ABB RAPID module: MainModule.mod

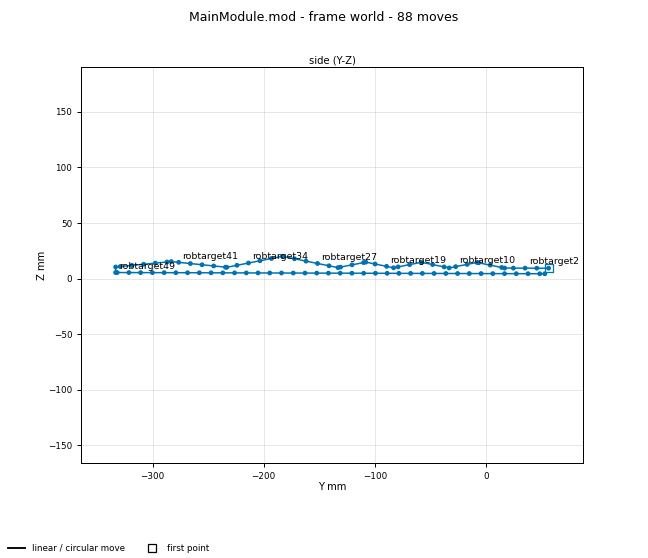
[picture p0: tool path of MainModule.mod in frame world, 88 of 89 moves have a stored position in this frame; points joined in program order, loops and branches not executed]
Module MainModule
!Declarations
!jointtarget
VAR jointtarget In:=[[7.408424,53.50812,4.795727,0.087915,31.638713,125.775488],[9E9,9E9,9E9,9E9,9E9,9E9]];

!robtarget
CONST robtarget robtarget0:=[[431.569187,56.285063,9.381984],[-0.000698,0.99784,0.064795,0.010754],[0,0,1,0],[9E9,9E9,9E9,9E9,9E9,9E9]];
CONST robtarget robtarget1:=[[431.569187,45.724144,9.412298],[-0.000572,0.998549,0.05275,0.010827],[0,0,1,0],[9E9,9E9,9E9,9E9,9E9,9E9]];
CONST robtarget robtarget2:=[[431.569187,35.163224,9.442612],[-0.000443,0.999115,0.040635,0.010893],[0,0,1,0],[9E9,9E9,9E9,9E9,9E9,9E9]];
CONST robtarget robtarget3:=[[431.569187,24.602305,9.472927],[-0.000312,0.999535,0.028467,0.010951],[0,0,1,0],[9E9,9E9,9E9,9E9,9E9,9E9]];
CONST robtarget robtarget4:=[[431.569187,16.862962,9.495142],[-0.000215,0.999749,0.019524,0.010988],[0,0,1,0],[9E9,9E9,9E9,9E9,9E9,9E9]];
CONST robtarget robtarget5:=[[431.569187,14.097751,10.056362],[-0.00019,0.999799,0.016325,0.011641],[0,-1,1,0],[9E9,9E9,9E9,9E9,9E9,9E9]];
CONST robtarget robtarget6:=[[431.569187,3.747803,12.15696],[-0.000061,0.999891,0.004342,0.01408],[0,-1,1,0],[9E9,9E9,9E9,9E9,9E9,9E9]];
CONST robtarget robtarget7:=[[431.569187,-6.602145,14.257559],[0.000126,0.999834,-0.007647,0.016509],[-1,0,1,0],[9E9,9E9,9E9,9E9,9E9,9E9]];
CONST robtarget robtarget8:=[[431.569187,-8.128353,14.567314],[0.000159,0.999813,-0.009415,0.016866],[-1,0,1,0],[9E9,9E9,9E9,9E9,9E9,9E9]];
CONST robtarget robtarget9:=[[431.569187,-16.962196,12.826988],[0.000292,0.999697,-0.019638,0.014842],[-1,0,1,0],[9E9,9E9,9E9,9E9,9E9,9E9]];
CONST robtarget robtarget10:=[[431.569187,-27.323994,10.785644],[0.000394,0.999423,-0.031607,0.012462],[-1,0,1,0],[9E9,9E9,9E9,9E9,9E9,9E9]];
CONST robtarget robtarget11:=[[431.569187,-33.145913,9.638687],[0.000427,0.999204,-0.038315,0.011124],[-1,0,1,0],[9E9,9E9,9E9,9E9,9E9,9E9]];
CONST robtarget robtarget12:=[[431.569187,-37.6806,10.559035],[0.00053,0.998978,-0.043528,0.012173],[-1,-1,1,0],[9E9,9E9,9E9,9E9,9E9,9E9]];
CONST robtarget robtarget13:=[[431.569187,-48.030548,12.659634],[0.000807,0.998359,-0.055384,0.01455],[-1,-1,1,0],[9E9,9E9,9E9,9E9,9E9,9E9]];
CONST robtarget robtarget14:=[[431.569187,-58.137228,14.71086],[0.00113,0.997617,-0.066893,0.016846],[-1,0,1,0],[9E9,9E9,9E9,9E9,9E9,9E9]];
CONST robtarget robtarget15:=[[431.569187,-58.380774,14.66288],[0.00113,0.9976,-0.06717,0.016789],[-1,0,1,0],[9E9,9E9,9E9,9E9,9E9,9E9]];
CONST robtarget robtarget16:=[[431.569187,-68.742572,12.621536],[0.001139,0.996779,-0.078889,0.014391],[-1,0,1,0],[9E9,9E9,9E9,9E9,9E9,9E9]];
CONST robtarget robtarget17:=[[431.569187,-79.10437,10.580192],[0.001091,0.995823,-0.090511,0.012005],[-1,0,1,0],[9E9,9E9,9E9,9E9,9E9,9E9]];
CONST robtarget robtarget18:=[[431.569187,-83.154788,9.782233],[0.001057,0.995413,-0.095024,0.011076],[-1,0,1,0],[9E9,9E9,9E9,9E9,9E9,9E9]];
CONST robtarget robtarget19:=[[431.569187,-89.45895,11.061709],[0.00128,0.994704,-0.102011,0.01248],[-1,-1,1,0],[9E9,9E9,9E9,9E9,9E9,9E9]];
CONST robtarget robtarget20:=[[431.569187,-99.808898,13.162308],[0.001684,0.993441,-0.11338,0.014757],[-1,-1,1,0],[9E9,9E9,9E9,9E9,9E9,9E9]];
CONST robtarget robtarget21:=[[431.569187,-108.146103,14.854406],[0.002043,0.992336,-0.122441,0.016561],[-1,0,1,0],[9E9,9E9,9E9,9E9,9E9,9E9]];
CONST robtarget robtarget22:=[[431.569187,-110.16115,14.457428],[0.002022,0.992072,-0.124619,0.016097],[-1,0,1,0],[9E9,9E9,9E9,9E9,9E9,9E9]];
CONST robtarget robtarget23:=[[431.569187,-120.522948,12.416084],[0.00188,0.990649,-0.135731,0.013723],[-1,0,1,0],[9E9,9E9,9E9,9E9,9E9,9E9]];
CONST robtarget robtarget24:=[[431.569187,-130.884746,10.37474],[0.001687,0.989116,-0.146689,0.011376],[-1,0,1,0],[9E9,9E9,9E9,9E9,9E9,9E9]];
CONST robtarget robtarget25:=[[431.569187,-133.163663,9.925778],[0.001638,0.988764,-0.149077,0.010864],[-1,0,1,0],[9E9,9E9,9E9,9E9,9E9,9E9]];
CONST robtarget robtarget26:=[[431.569187,-141.2373,11.564383],[0.002005,0.987442,-0.157468,0.012572],[-1,-1,1,0],[9E9,9E9,9E9,9E9,9E9,9E9]];
CONST robtarget robtarget27:=[[431.569187,-151.587248,13.664982],[0.00251,0.985662,-0.168072,0.01472],[-1,-1,1,0],[9E9,9E9,9E9,9E9,9E9,9E9]];
CONST robtarget robtarget28:=[[431.569187,-161.937196,15.76558],[0.003052,0.983792,-0.178497,0.016819],[-1,-1,1,0],[9E9,9E9,9E9,9E9,9E9,9E9]];
CONST robtarget robtarget29:=[[431.569187,-172.287145,17.866179],[0.003627,0.981839,-0.188739,0.018868],[-1,-1,1,0],[9E9,9E9,9E9,9E9,9E9,9E9]];
CONST robtarget robtarget30:=[[431.569187,-182.637093,19.966778],[0.004233,0.979811,-0.19879,0.020864],[-1,0,1,0],[9E9,9E9,9E9,9E9,9E9,9E9]];
CONST robtarget robtarget31:=[[431.569187,-183.146294,20.070124],[0.004264,0.979709,-0.19928,0.020961],[-1,0,1,0],[9E9,9E9,9E9,9E9,9E9,9E9]];
CONST robtarget robtarget32:=[[431.569187,-192.998307,18.129211],[0.004,0.977797,-0.208678,0.018741],[-1,0,1,0],[9E9,9E9,9E9,9E9,9E9,9E9]];
CONST robtarget robtarget33:=[[431.569187,-203.360105,16.087868],[0.003681,0.97572,-0.21837,0.016447],[-1,0,1,0],[9E9,9E9,9E9,9E9,9E9,9E9]];
CONST robtarget robtarget34:=[[431.569187,-213.721903,14.046524],[0.003322,0.973584,-0.227864,0.014195],[-1,0,1,0],[9E9,9E9,9E9,9E9,9E9,9E9]];
CONST robtarget robtarget35:=[[431.569187,-224.083701,12.00518],[0.002927,0.971393,-0.237157,0.011989],[-1,0,1,0],[9E9,9E9,9E9,9E9,9E9,9E9]];
CONST robtarget robtarget36:=[[431.569187,-233.181413,10.21287],[0.002552,0.96943,-0.245149,0.010091],[-1,0,1,0],[9E9,9E9,9E9,9E9,9E9,9E9]];
CONST robtarget robtarget37:=[[431.569187,-234.46303,10.344732],[0.002593,0.969146,-0.246261,0.010205],[-1,0,1,0],[9E9,9E9,9E9,9E9,9E9,9E9]];
CONST robtarget robtarget38:=[[431.569187,-244.968535,11.425619],[0.002938,0.966803,-0.255262,0.011128],[-1,-1,1,0],[9E9,9E9,9E9,9E9,9E9,9E9]];
CONST robtarget robtarget39:=[[431.569187,-255.474039,12.506506],[0.003292,0.964427,-0.264055,0.012023],[-1,0,1,0],[9E9,9E9,9E9,9E9,9E9,9E9]];
CONST robtarget robtarget40:=[[431.569187,-265.979544,13.587392],[0.003653,0.962023,-0.272641,0.01289],[-1,0,1,0],[9E9,9E9,9E9,9E9,9E9,9E9]];
CONST robtarget robtarget41:=[[431.569187,-276.485048,14.668279],[0.00402,0.959595,-0.281021,0.013728],[-1,0,1,0],[9E9,9E9,9E9,9E9,9E9,9E9]];
CONST robtarget robtarget42:=[[431.569187,-283.177166,15.356815],[0.004257,0.958039,-0.286252,0.014248],[-1,0,1,0],[9E9,9E9,9E9,9E9,9E9,9E9]];
CONST robtarget robtarget43:=[[431.569187,-286.99274,14.986344],[0.00418,0.957159,-0.289201,0.013835],[-1,0,1,0],[9E9,9E9,9E9,9E9,9E9,9E9]];
CONST robtarget robtarget44:=[[431.569187,-297.504272,13.965734],[0.003958,0.954726,-0.297187,0.012716],[-1,0,1,0],[9E9,9E9,9E9,9E9,9E9,9E9]];
CONST robtarget robtarget45:=[[431.569187,-308.015803,12.945123],[0.003722,0.952283,-0.304974,0.011623],[-1,0,1,0],[9E9,9E9,9E9,9E9,9E9,9E9]];
CONST robtarget robtarget46:=[[431.569187,-318.527335,11.924513],[0.003474,0.949832,-0.312563,0.010557],[-1,0,1,0],[9E9,9E9,9E9,9E9,9E9,9E9]];
CONST robtarget robtarget47:=[[431.569187,-329.038866,10.903902],[0.003214,0.947378,-0.319958,0.009516],[-1,0,1,0],[9E9,9E9,9E9,9E9,9E9,9E9]];
CONST robtarget robtarget48:=[[431.569187,-333.199163,10.499961],[0.003108,0.946407,-0.322833,0.009112],[-1,0,1,0],[9E9,9E9,9E9,9E9,9E9,9E9]];
CONST robtarget robtarget49:=[[431.569187,-333.212285,5.499561],[0.001628,0.946436,-0.322853,0.004773],[-1,0,1,0],[9E9,9E9,9E9,9E9,9E9,9E9]];
CONST robtarget robtarget50:=[[431.569187,-331.831606,5.495597],[0.001625,0.946759,-0.321902,0.004779],[-1,0,1,0],[9E9,9E9,9E9,9E9,9E9,9E9]];
CONST robtarget robtarget51:=[[431.569187,-321.270687,5.465283],[0.001597,0.949235,-0.314526,0.004821],[-1,0,1,0],[9E9,9E9,9E9,9E9,9E9,9E9]];
CONST robtarget robtarget52:=[[431.569187,-310.709767,5.434969],[0.001569,0.95171,-0.306955,0.004863],[-1,0,1,0],[9E9,9E9,9E9,9E9,9E9,9E9]];
CONST robtarget robtarget53:=[[431.569187,-300.148848,5.404655],[0.001538,0.954181,-0.299186,0.004905],[-1,0,1,0],[9E9,9E9,9E9,9E9,9E9,9E9]];
CONST robtarget robtarget54:=[[431.569187,-289.587928,5.374341],[0.001506,0.956643,-0.291217,0.004946],[-1,0,1,0],[9E9,9E9,9E9,9E9,9E9,9E9]];
CONST robtarget robtarget55:=[[431.569187,-279.027009,5.344027],[0.001472,0.959093,-0.283043,0.004987],[-1,0,1,0],[9E9,9E9,9E9,9E9,9E9,9E9]];
CONST robtarget robtarget56:=[[431.569187,-268.466089,5.313713],[0.001436,0.961526,-0.274664,0.005026],[-1,0,1,0],[9E9,9E9,9E9,9E9,9E9,9E9]];
CONST robtarget robtarget57:=[[431.569187,-257.90517,5.283399],[0.001398,0.963937,-0.266078,0.005065],[-1,0,1,0],[9E9,9E9,9E9,9E9,9E9,9E9]];
CONST robtarget robtarget58:=[[431.569187,-247.34425,5.253085],[0.001358,0.966322,-0.257283,0.005102],[-1,0,1,0],[9E9,9E9,9E9,9E9,9E9,9E9]];
CONST robtarget robtarget59:=[[431.569187,-236.783331,5.222771],[0.001317,0.968674,-0.248278,0.005139],[-1,0,1,0],[9E9,9E9,9E9,9E9,9E9,9E9]];
CONST robtarget robtarget60:=[[431.569187,-226.222411,5.192457],[0.001274,0.970989,-0.239063,0.005173],[-1,0,1,0],[9E9,9E9,9E9,9E9,9E9,9E9]];
CONST robtarget robtarget61:=[[431.569187,-215.661492,5.162143],[0.001229,0.973261,-0.229639,0.005207],[-1,0,1,0],[9E9,9E9,9E9,9E9,9E9,9E9]];
CONST robtarget robtarget62:=[[431.569187,-205.100572,5.131828],[0.001181,0.975484,-0.220006,0.005238],[-1,0,1,0],[9E9,9E9,9E9,9E9,9E9,9E9]];
CONST robtarget robtarget63:=[[431.569187,-194.539653,5.101514],[0.001132,0.977651,-0.210166,0.005268],[-1,0,1,0],[9E9,9E9,9E9,9E9,9E9,9E9]];
CONST robtarget robtarget64:=[[431.569187,-183.978733,5.0712],[0.001082,0.979756,-0.200123,0.005295],[-1,0,1,0],[9E9,9E9,9E9,9E9,9E9,9E9]];
CONST robtarget robtarget65:=[[431.569187,-173.417814,5.040886],[0.001029,0.981793,-0.189879,0.00532],[-1,0,1,0],[9E9,9E9,9E9,9E9,9E9,9E9]];
CONST robtarget robtarget66:=[[431.569187,-162.856894,5.010572],[0.000975,0.983754,-0.179439,0.005343],[-1,0,1,0],[9E9,9E9,9E9,9E9,9E9,9E9]];
CONST robtarget robtarget67:=[[431.569187,-152.295975,4.980258],[0.000918,0.985634,-0.168808,0.005363],[-1,0,1,0],[9E9,9E9,9E9,9E9,9E9,9E9]];
CONST robtarget robtarget68:=[[431.569187,-141.735055,4.949944],[0.000861,0.987425,-0.157993,0.00538],[-1,0,1,0],[9E9,9E9,9E9,9E9,9E9,9E9]];
CONST robtarget robtarget69:=[[431.569187,-131.174136,4.91963],[0.000802,0.989121,-0.147,0.005394],[-1,0,1,0],[9E9,9E9,9E9,9E9,9E9,9E9]];
CONST robtarget robtarget70:=[[431.569187,-120.613216,4.889316],[0.000741,0.990716,-0.135838,0.005405],[-1,0,1,0],[9E9,9E9,9E9,9E9,9E9,9E9]];
CONST robtarget robtarget71:=[[431.569187,-110.052297,4.859002],[0.000679,0.992203,-0.124516,0.005412],[-1,0,1,0],[9E9,9E9,9E9,9E9,9E9,9E9]];
CONST robtarget robtarget72:=[[431.569187,-99.491377,4.828688],[0.000616,0.993575,-0.113044,0.005416],[-1,0,1,0],[9E9,9E9,9E9,9E9,9E9,9E9]];
CONST robtarget robtarget73:=[[431.569187,-88.930458,4.798373],[0.000552,0.994827,-0.101433,0.005416],[-1,0,1,0],[9E9,9E9,9E9,9E9,9E9,9E9]];
CONST robtarget robtarget74:=[[431.569187,-78.369538,4.768059],[0.000487,0.995954,-0.089695,0.005413],[-1,0,1,0],[9E9,9E9,9E9,9E9,9E9,9E9]];
CONST robtarget robtarget75:=[[431.569187,-67.808619,4.737745],[0.000422,0.996951,-0.077843,0.005406],[-1,0,1,0],[9E9,9E9,9E9,9E9,9E9,9E9]];
CONST robtarget robtarget76:=[[431.569187,-57.247699,4.707431],[0.000356,0.997812,-0.065891,0.005395],[-1,0,1,0],[9E9,9E9,9E9,9E9,9E9,9E9]];
CONST robtarget robtarget77:=[[431.569187,-46.68678,4.677117],[0.00029,0.998534,-0.053853,0.005379],[-1,0,1,0],[9E9,9E9,9E9,9E9,9E9,9E9]];
CONST robtarget robtarget78:=[[431.569187,-36.12586,4.646803],[0.000224,0.999114,-0.041744,0.00536],[-1,0,1,0],[9E9,9E9,9E9,9E9,9E9,9E9]];
CONST robtarget robtarget79:=[[431.569187,-25.564941,4.616489],[0.000158,0.999548,-0.029579,0.005337],[-1,0,1,0],[9E9,9E9,9E9,9E9,9E9,9E9]];
CONST robtarget robtarget80:=[[431.569187,-15.004022,4.586175],[0.000092,0.999835,-0.017375,0.005309],[-1,0,1,0],[9E9,9E9,9E9,9E9,9E9,9E9]];
CONST robtarget robtarget81:=[[431.569187,-4.443102,4.555861],[0.000027,0.999973,-0.005147,0.005278],[-1,0,1,0],[9E9,9E9,9E9,9E9,9E9,9E9]];
CONST robtarget robtarget82:=[[431.569187,6.117817,4.525547],[-0.000037,0.999961,0.007087,0.005242],[0,0,1,0],[9E9,9E9,9E9,9E9,9E9,9E9]];
CONST robtarget robtarget83:=[[431.569187,16.678737,4.495233],[-0.000101,0.9998,0.019312,0.005203],[0,0,1,0],[9E9,9E9,9E9,9E9,9E9,9E9]];
CONST robtarget robtarget84:=[[431.569187,27.239656,4.464919],[-0.000163,0.99949,0.031511,0.00516],[0,0,1,0],[9E9,9E9,9E9,9E9,9E9,9E9]];
CONST robtarget robtarget85:=[[431.569187,37.800576,4.434604],[-0.000223,0.999033,0.043668,0.005113],[0,0,1,0],[9E9,9E9,9E9,9E9,9E9,9E9]];
CONST robtarget robtarget86:=[[431.569187,48.361495,4.40429],[-0.000283,0.998431,0.055767,0.005063],[0,0,1,0],[9E9,9E9,9E9,9E9,9E9,9E9]];
CONST robtarget robtarget87:=[[431.569187,52.881866,4.391315],[-0.000308,0.99813,0.060925,0.00504],[0,0,1,0],[9E9,9E9,9E9,9E9,9E9,9E9]];

!speeddata
VAR speeddata speeddata0:=[250,572.957795,5000,1000];

!tooldata
PERS tooldata ToolOfLove:=[True,[[0.015258,-0.149222,99.918848],[1,0,0,0]],[0.001,[0,0,0.1],[1,0,0,0],0,0,0]];

!wobjdata
PERS wobjdata Root:=[False,True,"",[[0,0,0],[1,0,0,0]],[[0,0,0],[1,0,0,0]]];

!zonedata
VAR zonedata zonedata0:=[False,1,5,1,5,1,5];

Proc Main()
ConfL \On;
ConfJ \On;
SingArea \Wrist;
MoveAbsJ In, speeddata0, zonedata0, ToolOfLove;
MoveL robtarget0, speeddata0, zonedata0, ToolOfLove \WObj:=Root;
MoveL robtarget1, speeddata0, zonedata0, ToolOfLove \WObj:=Root;
MoveL robtarget2, speeddata0, zonedata0, ToolOfLove \WObj:=Root;
MoveL robtarget3, speeddata0, zonedata0, ToolOfLove \WObj:=Root;
MoveL robtarget4, speeddata0, zonedata0, ToolOfLove \WObj:=Root;
MoveL robtarget5, speeddata0, zonedata0, ToolOfLove \WObj:=Root;
MoveL robtarget6, speeddata0, zonedata0, ToolOfLove \WObj:=Root;
MoveL robtarget7, speeddata0, zonedata0, ToolOfLove \WObj:=Root;
MoveL robtarget8, speeddata0, zonedata0, ToolOfLove \WObj:=Root;
MoveL robtarget9, speeddata0, zonedata0, ToolOfLove \WObj:=Root;
MoveL robtarget10, speeddata0, zonedata0, ToolOfLove \WObj:=Root;
MoveL robtarget11, speeddata0, zonedata0, ToolOfLove \WObj:=Root;
MoveL robtarget12, speeddata0, zonedata0, ToolOfLove \WObj:=Root;
MoveL robtarget13, speeddata0, zonedata0, ToolOfLove \WObj:=Root;
MoveL robtarget14, speeddata0, zonedata0, ToolOfLove \WObj:=Root;
MoveL robtarget15, speeddata0, zonedata0, ToolOfLove \WObj:=Root;
MoveL robtarget16, speeddata0, zonedata0, ToolOfLove \WObj:=Root;
MoveL robtarget17, speeddata0, zonedata0, ToolOfLove \WObj:=Root;
MoveL robtarget18, speeddata0, zonedata0, ToolOfLove \WObj:=Root;
MoveL robtarget19, speeddata0, zonedata0, ToolOfLove \WObj:=Root;
MoveL robtarget20, speeddata0, zonedata0, ToolOfLove \WObj:=Root;
MoveL robtarget21, speeddata0, zonedata0, ToolOfLove \WObj:=Root;
MoveL robtarget22, speeddata0, zonedata0, ToolOfLove \WObj:=Root;
MoveL robtarget23, speeddata0, zonedata0, ToolOfLove \WObj:=Root;
MoveL robtarget24, speeddata0, zonedata0, ToolOfLove \WObj:=Root;
MoveL robtarget25, speeddata0, zonedata0, ToolOfLove \WObj:=Root;
MoveL robtarget26, speeddata0, zonedata0, ToolOfLove \WObj:=Root;
MoveL robtarget27, speeddata0, zonedata0, ToolOfLove \WObj:=Root;
MoveL robtarget28, speeddata0, zonedata0, ToolOfLove \WObj:=Root;
MoveL robtarget29, speeddata0, zonedata0, ToolOfLove \WObj:=Root;
MoveL robtarget30, speeddata0, zonedata0, ToolOfLove \WObj:=Root;
MoveL robtarget31, speeddata0, zonedata0, ToolOfLove \WObj:=Root;
MoveL robtarget32, speeddata0, zonedata0, ToolOfLove \WObj:=Root;
MoveL robtarget33, speeddata0, zonedata0, ToolOfLove \WObj:=Root;
MoveL robtarget34, speeddata0, zonedata0, ToolOfLove \WObj:=Root;
MoveL robtarget35, speeddata0, zonedata0, ToolOfLove \WObj:=Root;
MoveL robtarget36, speeddata0, zonedata0, ToolOfLove \WObj:=Root;
MoveL robtarget37, speeddata0, zonedata0, ToolOfLove \WObj:=Root;
MoveL robtarget38, speeddata0, zonedata0, ToolOfLove \WObj:=Root;
MoveL robtarget39, speeddata0, zonedata0, ToolOfLove \WObj:=Root;
MoveL robtarget40, speeddata0, zonedata0, ToolOfLove \WObj:=Root;
MoveL robtarget41, speeddata0, zonedata0, ToolOfLove \WObj:=Root;
MoveL robtarget42, speeddata0, zonedata0, ToolOfLove \WObj:=Root;
MoveL robtarget43, speeddata0, zonedata0, ToolOfLove \WObj:=Root;
MoveL robtarget44, speeddata0, zonedata0, ToolOfLove \WObj:=Root;
MoveL robtarget45, speeddata0, zonedata0, ToolOfLove \WObj:=Root;
MoveL robtarget46, speeddata0, zonedata0, ToolOfLove \WObj:=Root;
MoveL robtarget47, speeddata0, zonedata0, ToolOfLove \WObj:=Root;
MoveL robtarget48, speeddata0, zonedata0, ToolOfLove \WObj:=Root;
MoveL robtarget49, speeddata0, zonedata0, ToolOfLove \WObj:=Root;
MoveL robtarget50, speeddata0, zonedata0, ToolOfLove \WObj:=Root;
MoveL robtarget51, speeddata0, zonedata0, ToolOfLove \WObj:=Root;
MoveL robtarget52, speeddata0, zonedata0, ToolOfLove \WObj:=Root;
MoveL robtarget53, speeddata0, zonedata0, ToolOfLove \WObj:=Root;
MoveL robtarget54, speeddata0, zonedata0, ToolOfLove \WObj:=Root;
MoveL robtarget55, speeddata0, zonedata0, ToolOfLove \WObj:=Root;
MoveL robtarget56, speeddata0, zonedata0, ToolOfLove \WObj:=Root;
MoveL robtarget57, speeddata0, zonedata0, ToolOfLove \WObj:=Root;
MoveL robtarget58, speeddata0, zonedata0, ToolOfLove \WObj:=Root;
MoveL robtarget59, speeddata0, zonedata0, ToolOfLove \WObj:=Root;
MoveL robtarget60, speeddata0, zonedata0, ToolOfLove \WObj:=Root;
MoveL robtarget61, speeddata0, zonedata0, ToolOfLove \WObj:=Root;
MoveL robtarget62, speeddata0, zonedata0, ToolOfLove \WObj:=Root;
MoveL robtarget63, speeddata0, zonedata0, ToolOfLove \WObj:=Root;
MoveL robtarget64, speeddata0, zonedata0, ToolOfLove \WObj:=Root;
MoveL robtarget65, speeddata0, zonedata0, ToolOfLove \WObj:=Root;
MoveL robtarget66, speeddata0, zonedata0, ToolOfLove \WObj:=Root;
MoveL robtarget67, speeddata0, zonedata0, ToolOfLove \WObj:=Root;
MoveL robtarget68, speeddata0, zonedata0, ToolOfLove \WObj:=Root;
MoveL robtarget69, speeddata0, zonedata0, ToolOfLove \WObj:=Root;
MoveL robtarget70, speeddata0, zonedata0, ToolOfLove \WObj:=Root;
MoveL robtarget71, speeddata0, zonedata0, ToolOfLove \WObj:=Root;
MoveL robtarget72, speeddata0, zonedata0, ToolOfLove \WObj:=Root;
MoveL robtarget73, speeddata0, zonedata0, ToolOfLove \WObj:=Root;
MoveL robtarget74, speeddata0, zonedata0, ToolOfLove \WObj:=Root;
MoveL robtarget75, speeddata0, zonedata0, ToolOfLove \WObj:=Root;
MoveL robtarget76, speeddata0, zonedata0, ToolOfLove \WObj:=Root;
MoveL robtarget77, speeddata0, zonedata0, ToolOfLove \WObj:=Root;
MoveL robtarget78, speeddata0, zonedata0, ToolOfLove \WObj:=Root;
MoveL robtarget79, speeddata0, zonedata0, ToolOfLove \WObj:=Root;
MoveL robtarget80, speeddata0, zonedata0, ToolOfLove \WObj:=Root;
MoveL robtarget81, speeddata0, zonedata0, ToolOfLove \WObj:=Root;
MoveL robtarget82, speeddata0, zonedata0, ToolOfLove \WObj:=Root;
MoveL robtarget83, speeddata0, zonedata0, ToolOfLove \WObj:=Root;
MoveL robtarget84, speeddata0, zonedata0, ToolOfLove \WObj:=Root;
MoveL robtarget85, speeddata0, zonedata0, ToolOfLove \WObj:=Root;
MoveL robtarget86, speeddata0, zonedata0, ToolOfLove \WObj:=Root;
MoveL robtarget87, speeddata0, zonedata0, ToolOfLove \WObj:=Root;
EndProc
EndModule
